Universal Robots PolyScope program: proj1_final.urp

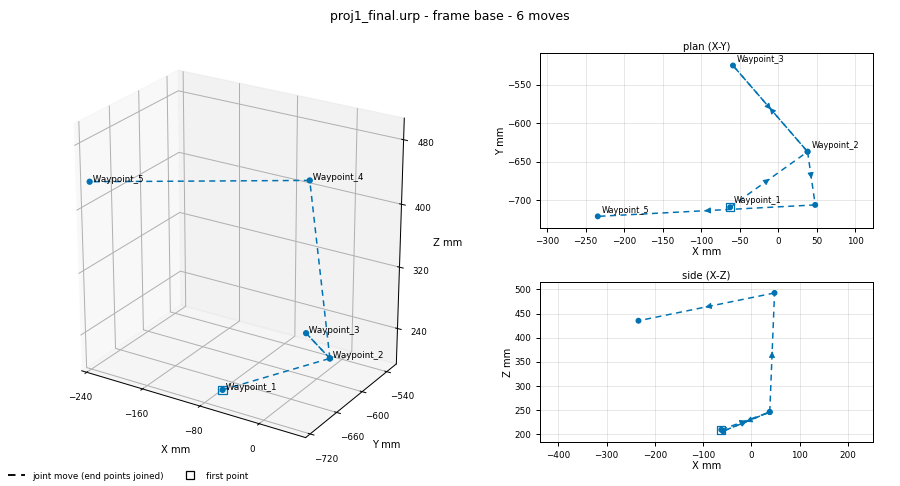
[picture p0: tool path of proj1_final.urp in frame base, 6 of 6 moves have a stored position in this frame; points joined in program order, loops and branches not executed]
Program proj1_final (installation=default directory=/programs/usbdisk/project1_final createdIn=5.11.10.1010502 lastSavedIn=5.11.10.1010502 robotSerialNumber=20225201357)
Calibrated DH parameters: a=[-0.000097, -0.065329, -0.560646, 0.000001, -0.00004, 0]; d=[0.180831, -263.113709, 285.24385, -21.955837, 0.119737, 0.115719]; alpha=[1.571643, -0.002312, 0.004975, 1.569542, -1.570894, 0]; deltaTheta=[0, 1.463798, 5.013296, -0.193909, 0, 0]
Robot Program (runOnlyOnce=true)
  MoveJ speed 60 deg/s, acceleration 80 deg/s^2 (useActiveTCP=true) feature=Base
    Waypoint Waypoint_1: motionParameters(nextMotionTime=3); TCP in base x=-62.466 y=-708.919 z=209.481 mm, rx=-1.6329 ry=2.6091 rz=0.0797 rad; joints [72.85, -84.804, 105.655, -107.692, 269.15, -17.56] deg; TCP offset x=20.709 y=-1.468 z=254.962 mm, rx=-0.0022 ry=-0.0343 rz=-1.1076 rad
    Waypoint Waypoint_2: motionParameters(nextMotionTime=3); TCP in base x=37.905 y=-636.981 z=246.056 mm, rx=-1.7471 ry=2.5382 rz=0.0855 rad; joints [79.872, -92.925, 110.074, -103.97, 269.177, -15.54] deg
    Waypoint Waypoint_3: motionParameters(nextMotionTime=3); TCP in base x=-58.814 y=-525.231 z=206.359 mm, rx=-1.9792 ry=2.3236 rz=0.1346 rad; joints [67.888, -102.346, 121.965, -104.693, 267.505, -39.194] deg
    Waypoint Waypoint_2: motionParameters(nextMotionTime=3); TCP in base x=37.905 y=-636.981 z=246.056 mm, rx=-1.7471 ry=2.5382 rz=0.0855 rad; joints [79.872, -92.925, 110.074, -103.97, 269.177, -15.54] deg
    Waypoint Waypoint_4: motionParameters(nextMotionTime=3); TCP in base x=47.813 y=-705.961 z=492.852 mm, rx=-1.5112 ry=2.2362 rz=-0.1791 rad; joints [70.335, -85.601, 77.642, -67.342, 289.9, -26.654] deg
    Waypoint Waypoint_5: motionParameters(nextMotionTime=4); TCP in base x=-234.122 y=-720.797 z=435.231 mm, rx=-1.306 ry=1.8617 rz=-0.4789 rad; joints [45.406, -67.02, 64.373, -43.101, 297.952, -62.294] deg
